// TIA Portal project "vize" (V15.1)

(* hardware
DEVICE "S7-1200 station_1"  S7-1200 Station
   slot 0: "Rack_0"  S7-1200 Rack  Rack  V1.0
   slot 1: "PLC_1"  CPU 1214C DC/DC/DC  6ES7 214-1AG40-0XB0  V4.2
*)

// ===== PLC "PLC_1"  CPU 1214C DC/DC/DC =====

VAR_GLOBAL   // PLC tag table "Default tag table"
   "General_Start" AT %M0.0 : Bool;
   "Reset_and_Start" AT %Q0.0 : Bool;
   "Start_Control_Loop" AT %Q0.1 : Bool;
   "Time_End" AT %M0.1 : Bool;
END_VAR

DATA_BLOCK "general_memory"   // DB1
{ S7_Optimized_Access := 'TRUE' }
VERSION : 0.1
   VAR RETAIN
      x1_data : Array[0..500] of Real;
      x2_data : Array[0..500] of Real;
      u_data : Array[0..500] of Real;
   END_VAR
BEGIN
END_DATA_BLOCK

DATA_BLOCK "Initial_values_DB"   // DB2
{ S7_Optimized_Access := 'TRUE' }
VERSION : 0.1
// stored: InstanceOfName Initial_values
"Initial_values"
BEGIN
END_DATA_BLOCK

DATA_BLOCK "System_Integration_DB"   // DB4
{ S7_Optimized_Access := 'TRUE' }
VERSION : 0.1
// stored: InstanceOfName System_Integration
"System_Integration"
BEGIN
END_DATA_BLOCK

DATA_BLOCK "Startup_DB"   // DB5
{ S7_Optimized_Access := 'TRUE' }
VERSION : 0.1
   VAR RETAIN
      startup_counter : Int;
   END_VAR
BEGIN
END_DATA_BLOCK

// folder: System blocks/Program resources

DATA_BLOCK "General_Timer"   // DB3
{ S7_Optimized_Access := 'TRUE' }
AUTHOR : Simatic
FAMILY : IEC
NAME : IEC_TMR
VERSION : 1.0
// stored: InstanceOfName IEC_TIMER
"IEC_TIMER"
BEGIN
END_DATA_BLOCK

// folder: (top level)

FUNCTION_BLOCK "Initial_values"   // FB1, LAD
{ S7_Optimized_Access := 'TRUE' }
VERSION : 0.1
   VAR_INPUT
      start : Bool;
   END_VAR
BEGIN

REGION Network 1
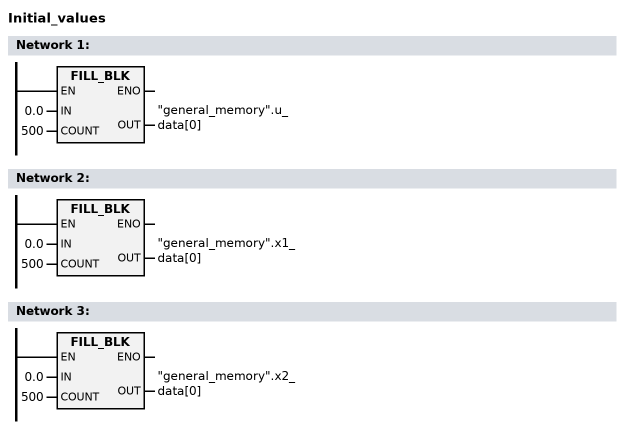
   RUNG wire#powerrail
      FillBlockI(in := 0.0, count := 500, out => "general_memory".u_data[0])
   END_RUNG
   // the same network as SCL:
   FILL_BLK(IN := 0.0, COUNT := 500, OUT => "general_memory".u_data[0]);
END_REGION

REGION Network 2
   RUNG wire#powerrail
      FillBlockI(in := 0.0, count := 500, out => "general_memory".x1_data[0])
   END_RUNG
   // the same network as SCL:
   FILL_BLK(IN := 0.0, COUNT := 500, OUT => "general_memory".x1_data[0]);
END_REGION

REGION Network 3
   RUNG wire#powerrail
      FillBlockI(in := 0.0, count := 500, out => "general_memory".x2_data[0])
   END_RUNG
   // the same network as SCL:
   FILL_BLK(IN := 0.0, COUNT := 500, OUT => "general_memory".x2_data[0]);
END_REGION
END_FUNCTION_BLOCK

FUNCTION_BLOCK "System_Integration"   // FB2, LAD
{ S7_Optimized_Access := 'TRUE' }
VERSION : 0.1
   VAR_INPUT
      Start_Control_Loop : Bool;
   END_VAR
   VAR
      pozitif_kenar : Bool;
      k : Int;
      "k+1" : Int;
      "k-1" : Int;
      x1temp : Array[0..500] of Real;
      x2temp : Array[0..500] of Real;
      xref1 : Array[0..500] of Real;
      xref2 : Array[0..500] of Real;
      xrefdot_1 : Array[0..500] of Real;
      xrefdot_2 : Array[0..500] of Real;
      error1 : Array[0..500] of Real;
      error2 : Array[0..500] of Real;
      surface : Array[0..500] of Real;
      "abs(surface)" : Real;
      sat : Array[0..500] of Real;
      fhat : Array[0..500] of Real;
      dot_deriv : Array[0..500] of Real;
      uk : Array[0..500] of Real;
      minus_fhat : Real;
      xdot_1 : Array[0..500] of Real;
      xdot_2 : Array[0..500] of Real;
   END_VAR
   VAR CONSTANT
      cc : Real := 1.0;
      ww : Real := 2.0;
      aa : Real := 2.5;
      umax : Real := 12.0;
      ks : Real := 0.1;
      lamda : Real := 50.0;
      thres : Real := 0.1;
      ts : Real := 0.001;
      a11 : Real;
      a12 : Real := 1.0;
      a21 : Real := -3.0;
      a22 : Real := -2.0;
      b21 : Real := 3.0;
      c11 : Real := 0.0;
      c12 : Real := 2.0;
   END_VAR
   VAR_TEMP   // added for the SCL form of the ladder/FBD networks
      _w1 : Bool;
   END_VAR
BEGIN

REGION Network 1
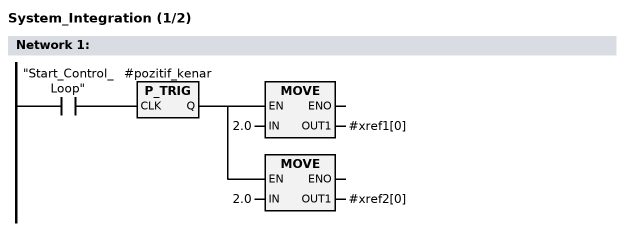
   RUNG wire#powerrail
      Contact( "Start_Control_Loop" )
      P_Trig( #pozitif_kenar )
      wire#w1
      Move(in := 2.0, out1 => #xref1[0])
   END_RUNG
   RUNG wire#w1
      Move(in := 2.0, out1 => #xref2[0])
   END_RUNG
   // the same network as SCL:
   #_w1 := "Start_Control_Loop" AND NOT #pozitif_kenar;   // rising edge
   #pozitif_kenar := "Start_Control_Loop";
   IF #_w1 THEN
       #xref1[0] := 2.0;
       #xref2[0] := 2.0;
   END_IF;
END_REGION

REGION Network 2
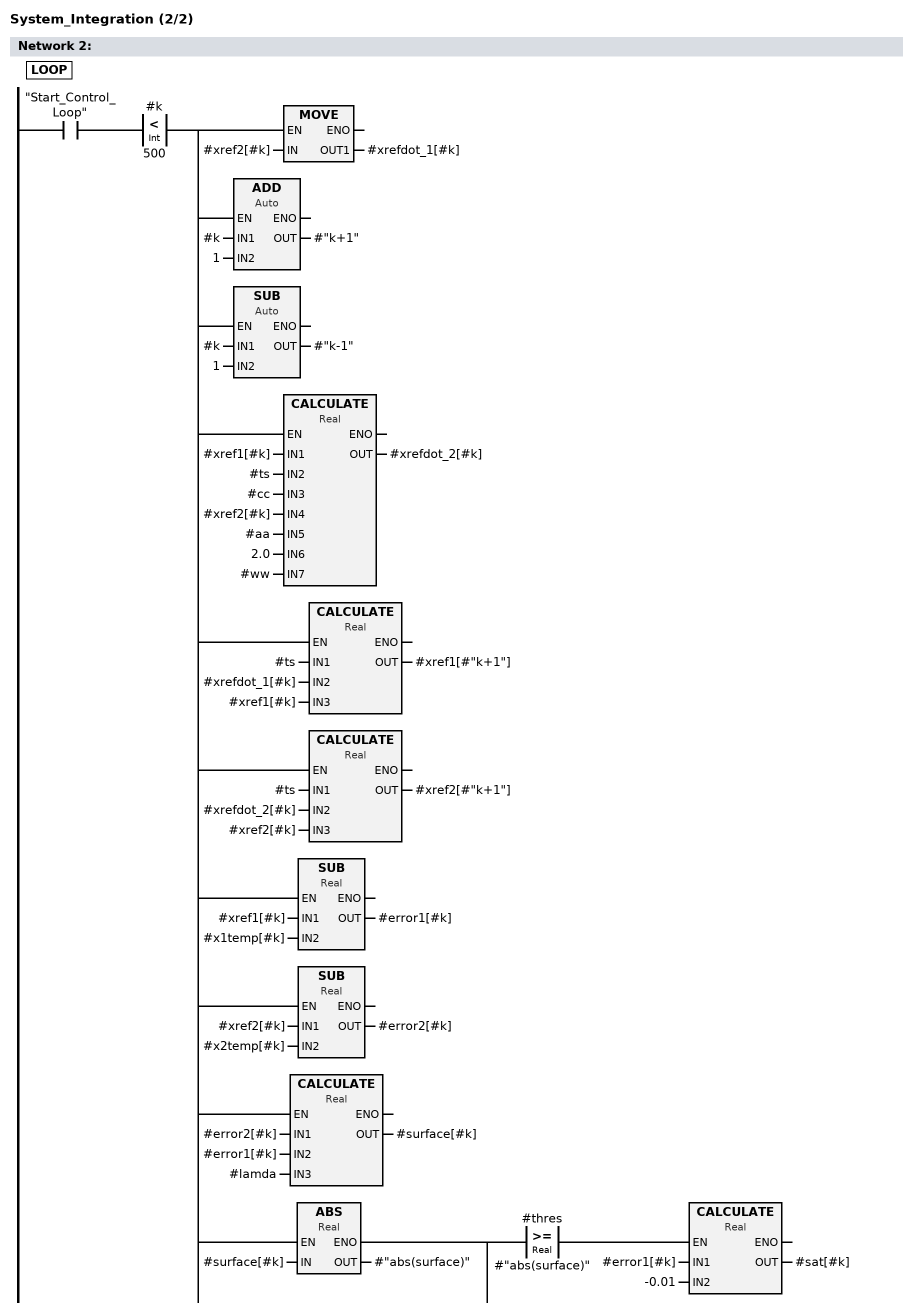
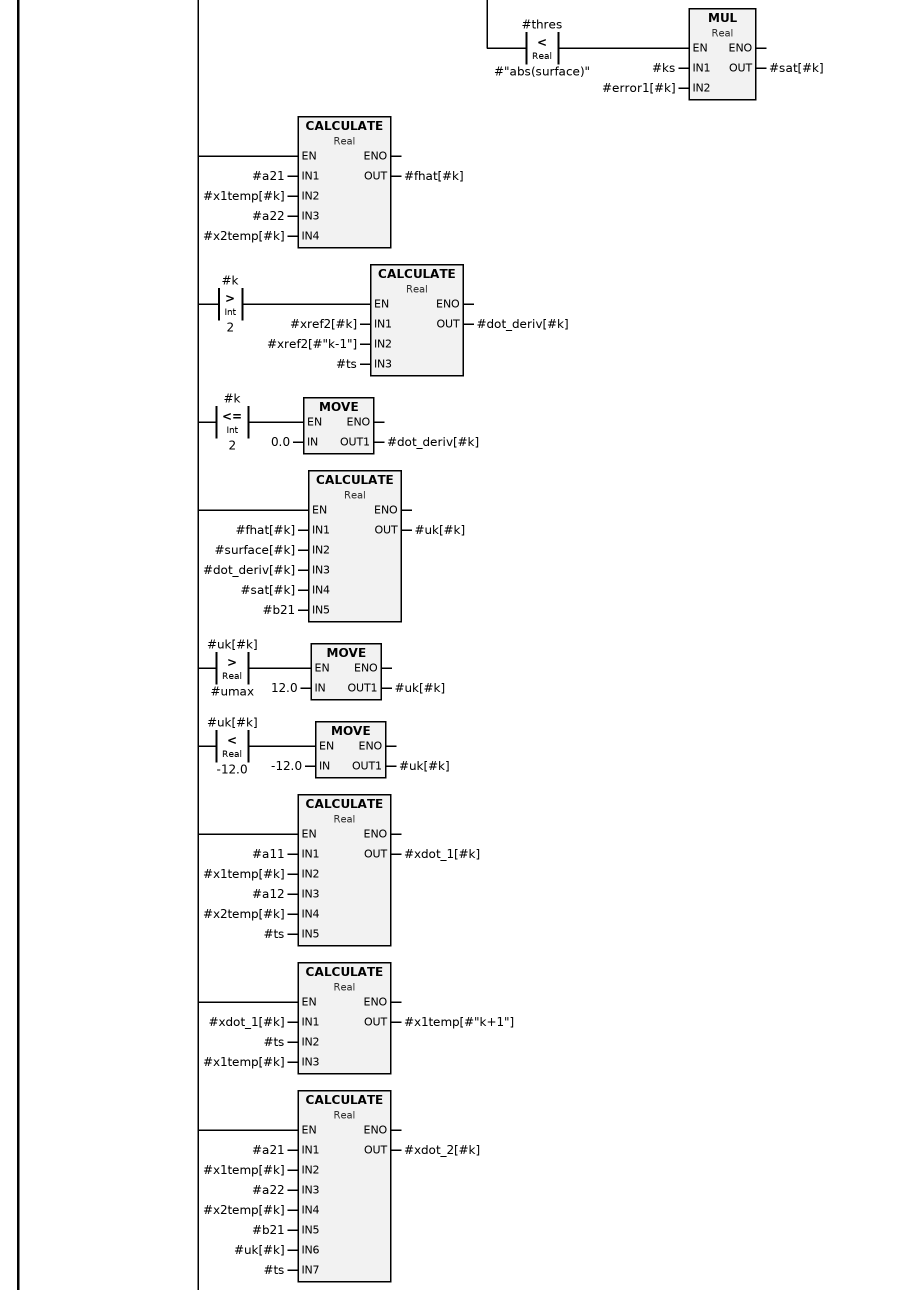
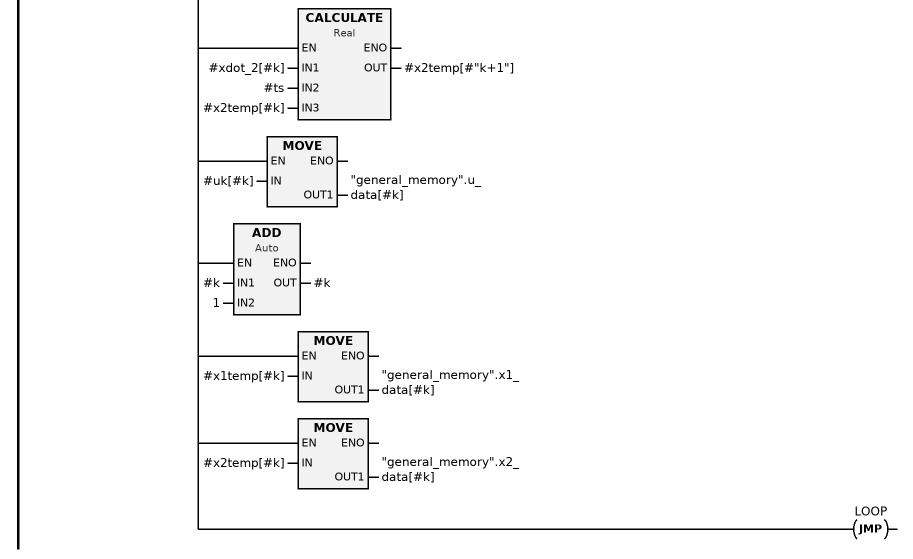
   Label( LOOP )
   RUNG wire#powerrail
      Contact( "Start_Control_Loop" )
      { S7_Templates := "SrcType := Int" } LT_Contact(in1 := #k, in2 := 500)
      wire#w1
      Move(in := #xref2[#k], out1 => #xrefdot_1[#k])
   END_RUNG
   RUNG wire#w1
      Add(in1 := #k, in2 := 1, out => #"k+1")
   END_RUNG
   RUNG wire#w1
      Sub(in1 := #k, in2 := 1, out => #"k-1")
   END_RUNG
   RUNG wire#w1
      { S7_Templates := "SrcType := Real"; S7_Expression := "IN3*(IN3-IN1**IN6)*IN4-IN1+IN5*COS(IN7)" } Calculate(in1 := #xref1[#k], in2 := #ts, in3 := #cc, in4 := #xref2[#k], in5 := #aa, in6 := 2.0, in7 := #ww, out => #xrefdot_2[#k])
   END_RUNG
   RUNG wire#w1
      { S7_Templates := "SrcType := Real"; S7_Expression := "IN1*IN2+IN3" } Calculate(in1 := #ts, in2 := #xrefdot_1[#k], in3 := #xref1[#k], out => #xref1[#"k+1"])
   END_RUNG
   RUNG wire#w1
      { S7_Templates := "SrcType := Real"; S7_Expression := "IN1*IN2+IN3" } Calculate(in1 := #ts, in2 := #xrefdot_2[#k], in3 := #xref2[#k], out => #xref2[#"k+1"])
   END_RUNG
   RUNG wire#w1
      { S7_Templates := "SrcType := Real" } Sub(in1 := #xref1[#k], in2 := #x1temp[#k], out => #error1[#k])
   END_RUNG
   RUNG wire#w1
      { S7_Templates := "SrcType := Real" } Sub(in1 := #xref2[#k], in2 := #x2temp[#k], out => #error2[#k])
   END_RUNG
   RUNG wire#w1
      { S7_Templates := "SrcType := Real"; S7_Expression := "IN1+IN2*IN3" } Calculate(in1 := #error2[#k], in2 := #error1[#k], in3 := #lamda, out => #surface[#k])
   END_RUNG
   RUNG wire#w1
      { S7_Templates := "SrcType := Real" } Abs(in := #surface[#k], out => #"abs(surface)")
      wire#w2
      { S7_Templates := "SrcType := Real" } GE_Contact(in1 := #thres, in2 := #"abs(surface)")
      { S7_Templates := "SrcType := Real"; S7_Expression := "TAN(IN1)*IN2" } Calculate(in1 := #error1[#k], in2 := -0.01, out => #sat[#k])
   END_RUNG
   RUNG wire#w2
      { S7_Templates := "SrcType := Real" } LT_Contact(in1 := #thres, in2 := #"abs(surface)")
      { S7_Templates := "SrcType := Real" } Mul(in1 := #ks, in2 := #error1[#k], out => #sat[#k])
   END_RUNG
   RUNG wire#w1
      { S7_Templates := "SrcType := Real"; S7_Expression := "IN1*IN2+IN3*IN4" } Calculate(in1 := #a21, in2 := #x1temp[#k], in3 := #a22, in4 := #x2temp[#k], out => #fhat[#k])
   END_RUNG
   RUNG wire#w1
      { S7_Templates := "SrcType := Int" } GT_Contact(in1 := #k, in2 := 2)
      { S7_Templates := "SrcType := Real"; S7_Expression := "(IN1-IN2)/IN3" } Calculate(in1 := #xref2[#k], in2 := #xref2[#"k-1"], in3 := #ts, out => #dot_deriv[#k])
   END_RUNG
   RUNG wire#w1
      { S7_Templates := "SrcType := Int" } LE_Contact(in1 := #k, in2 := 2)
      Move(in := 0.0, out1 => #dot_deriv[#k])
   END_RUNG
   RUNG wire#w1
      { S7_Templates := "SrcType := Real"; S7_Expression := "(-IN1+IN2+IN3+IN4)/IN5" } Calculate(in1 := #fhat[#k], in2 := #surface[#k], in3 := #dot_deriv[#k], in4 := #sat[#k], in5 := #b21, out => #uk[#k])
   END_RUNG
   RUNG wire#w1
      { S7_Templates := "SrcType := Real" } GT_Contact(in1 := #uk[#k], in2 := #umax)
      Move(in := 12.0, out1 => #uk[#k])
   END_RUNG
   RUNG wire#w1
      { S7_Templates := "SrcType := Real" } LT_Contact(in1 := #uk[#k], in2 := -12.0)
      Move(in := -12.0, out1 => #uk[#k])
   END_RUNG
   RUNG wire#w1
      { S7_Templates := "SrcType := Real"; S7_Expression := "IN1*IN2+IN3*IN4" } Calculate(in1 := #a11, in2 := #x1temp[#k], in3 := #a12, in4 := #x2temp[#k], in5 := #ts, out => #xdot_1[#k])
   END_RUNG
   RUNG wire#w1
      { S7_Templates := "SrcType := Real"; S7_Expression := "IN1*IN2+IN3" } Calculate(in1 := #xdot_1[#k], in2 := #ts, in3 := #x1temp[#k], out => #x1temp[#"k+1"])
   END_RUNG
   RUNG wire#w1
      { S7_Templates := "SrcType := Real"; S7_Expression := "IN1*IN2+IN3*IN4+IN5*IN6" } Calculate(in1 := #a21, in2 := #x1temp[#k], in3 := #a22, in4 := #x2temp[#k], in5 := #b21, in6 := #uk[#k], in7 := #ts, out => #xdot_2[#k])
   END_RUNG
   RUNG wire#w1
      { S7_Templates := "SrcType := Real"; S7_Expression := "IN1*IN2+IN3" } Calculate(in1 := #xdot_2[#k], in2 := #ts, in3 := #x2temp[#k], out => #x2temp[#"k+1"])
   END_RUNG
   RUNG wire#w1
      Move(in := #uk[#k], out1 => "general_memory".u_data[#k])
   END_RUNG
   RUNG wire#w1
      Add(in1 := #k, in2 := 1, out => #k)
   END_RUNG
   RUNG wire#w1
      Move(in := #x1temp[#k], out1 => "general_memory".x1_data[#k])
   END_RUNG
   RUNG wire#w1
      Move(in := #x2temp[#k], out1 => "general_memory".x2_data[#k])
   END_RUNG
   RUNG wire#w1
      JumpCoil( LOOP )
   END_RUNG
   // the same network as SCL:
   LOOP:
   #_w1 := "Start_Control_Loop" AND (#k < 500);
   IF #_w1 THEN
       #xrefdot_1[#k] := #xref2[#k];
       #"k+1" := #k + 1;
       #"k-1" := #k - 1;
       #xrefdot_2[#k] := #cc*(#cc-#xref1[#k]**2.0)*#xref2[#k]-#xref1[#k]+#aa*COS(#ww);
       #xref1[#"k+1"] := #ts*#xrefdot_1[#k]+#xref1[#k];
       #xref2[#"k+1"] := #ts*#xrefdot_2[#k]+#xref2[#k];
       #error1[#k] := #xref1[#k] - #x1temp[#k];
       #error2[#k] := #xref2[#k] - #x2temp[#k];
       #surface[#k] := #error2[#k]+#error1[#k]*#lamda;
       #"abs(surface)" := ABS(#surface[#k]);
   END_IF;
   IF #_w1 AND (#thres >= #"abs(surface)") THEN #sat[#k] := TAN(#error1[#k])*(-0.01); END_IF;
   IF #_w1 AND (#thres < #"abs(surface)") THEN #sat[#k] := #ks * #error1[#k]; END_IF;
   IF #_w1 THEN #fhat[#k] := #a21*#x1temp[#k]+#a22*#x2temp[#k]; END_IF;
   IF #_w1 AND (#k > 2) THEN #dot_deriv[#k] := (#xref2[#k]-#xref2[#"k-1"])/#ts; END_IF;
   IF #_w1 AND (#k <= 2) THEN #dot_deriv[#k] := 0.0; END_IF;
   IF #_w1 THEN #uk[#k] := (-#fhat[#k]+#surface[#k]+#dot_deriv[#k]+#sat[#k])/#b21; END_IF;
   IF #_w1 AND (#uk[#k] > #umax) THEN #uk[#k] := 12.0; END_IF;
   IF #_w1 AND (#uk[#k] < (-12.0)) THEN #uk[#k] := -12.0; END_IF;
   IF #_w1 THEN
       #xdot_1[#k] := #a11*#x1temp[#k]+#a12*#x2temp[#k];
       #x1temp[#"k+1"] := #xdot_1[#k]*#ts+#x1temp[#k];
       #xdot_2[#k] := #a21*#x1temp[#k]+#a22*#x2temp[#k]+#b21*#uk[#k];
       #x2temp[#"k+1"] := #xdot_2[#k]*#ts+#x2temp[#k];
       "general_memory".u_data[#k] := #uk[#k];
       #k := #k + 1;
       "general_memory".x1_data[#k] := #x1temp[#k];
       "general_memory".x2_data[#k] := #x2temp[#k];
       GOTO LOOP;
   END_IF;
END_REGION
END_FUNCTION_BLOCK

ORGANIZATION_BLOCK "Main"   // OB1, LAD, ProgramCycle
TITLE = "Main Program Sweep (Cycle)"
{ S7_Optimized_Access := 'TRUE' }
VERSION : 0.1
   VAR_INPUT
      Initial_Call : Bool;   // Initial call of this OB
      Remanence : Bool;   // =True, if remanent data are available
   END_VAR
   VAR_TEMP   // added for the SCL form of the ladder/FBD networks
      _w1 : Bool;
   END_VAR
BEGIN

REGION Network 1
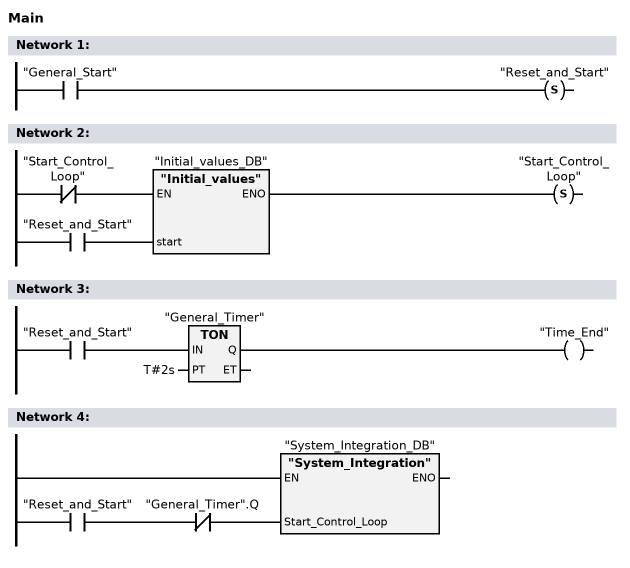
   RUNG wire#powerrail
      Contact( "General_Start" )
      S_Coil( "Reset_and_Start" )
   END_RUNG
   // the same network as SCL:
   IF "General_Start" THEN "Reset_and_Start" := TRUE; END_IF;
END_REGION

REGION Network 2
   RUNG wire#powerrail
      I_Contact( "Start_Control_Loop" )
      "Initial_values_DB"(start := wire#w1)
      S_Coil( "Start_Control_Loop" )
   END_RUNG
   RUNG wire#powerrail
      Contact( "Reset_and_Start" )
   END_RUNG wire#w1
   // the same network as SCL:
   "Initial_values_DB"(EN := NOT "Start_Control_Loop", start := "Reset_and_Start", ENO => #_w1);   // "Initial_values"
   IF #_w1 THEN "Start_Control_Loop" := TRUE; END_IF;
END_REGION

REGION Network 3
   "General_Timer".TON(IN := "Reset_and_Start", PT := T#2s);
   "Time_End" := "General_Timer".Q;
END_REGION

REGION Network 4
   RUNG wire#powerrail
      "System_Integration_DB"(Start_Control_Loop := wire#w1)
   END_RUNG
   RUNG wire#powerrail
      Contact( "Reset_and_Start" )
      I_Contact( "General_Timer".Q )
   END_RUNG wire#w1
   // the same network as SCL:
   "System_Integration_DB"(Start_Control_Loop := "Reset_and_Start" AND NOT "General_Timer".Q);   // "System_Integration"
END_REGION
END_ORGANIZATION_BLOCK

ORGANIZATION_BLOCK "Startup"   // OB100, LAD, Startup
TITLE = "Complete Restart"
{ S7_Optimized_Access := 'TRUE' }
VERSION : 0.1
   VAR_INPUT
      LostRetentive : Bool;   // True if retentive data are lost
      LostRTC : Bool;   // True if date and time are lost
   END_VAR
BEGIN

REGION Network 1
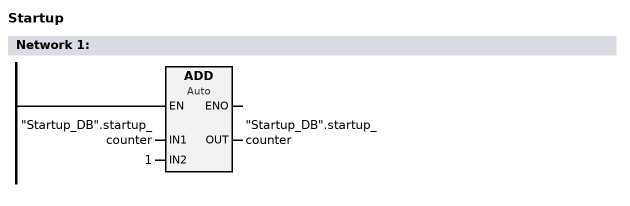
   RUNG wire#powerrail
      Add(in1 := "Startup_DB".startup_counter, in2 := 1, out => "Startup_DB".startup_counter)
   END_RUNG
   // the same network as SCL:
   "Startup_DB".startup_counter := "Startup_DB".startup_counter + 1;
END_REGION
END_ORGANIZATION_BLOCK